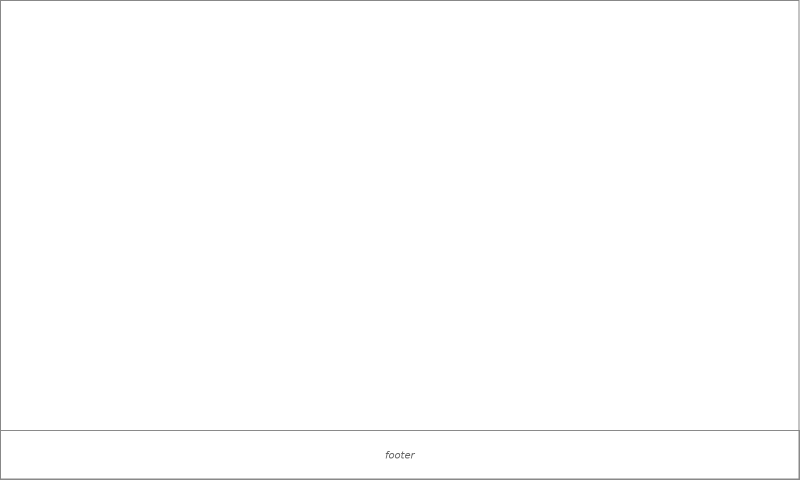
VISUALIZATION Group  // 800x480
    Frame (0,430 800x50)
        shows footer()
END_VISUALIZATION

(* stored: Version 1.1.0.1, ProductVersion 3.1.4024.12
   Visu Group: Id {e4707c97-ebc9-41f8-84d3-ae41a9611718} *)
